// TIA Portal V18 export
ORGANIZATION_BLOCK "10-Main"   // OB1, LAD, ProgramCycle
TITLE = "Main Program / "Main Program Sweep (Cycle)"
{ S7_Optimized_Access := 'TRUE' }
VERSION : 0.1
// stored: AutoNumber true, IsIECCheckEnabled false, SetENOAutomatically false
   VAR_INPUT
      Initial_Call : Bool;   // Initial call of this OB
      Remanence : Bool;   // =True, if remanent data are available
   END_VAR
   VAR_TEMP
      "Temp NormScale" : Real;
      Temp_1 : Bool;
      Temp_2 : Bool;
      "read date val" : DTL;
      "read date out" : Int;
   END_VAR
BEGIN

REGION Network 1: Off, On, Auto Definition
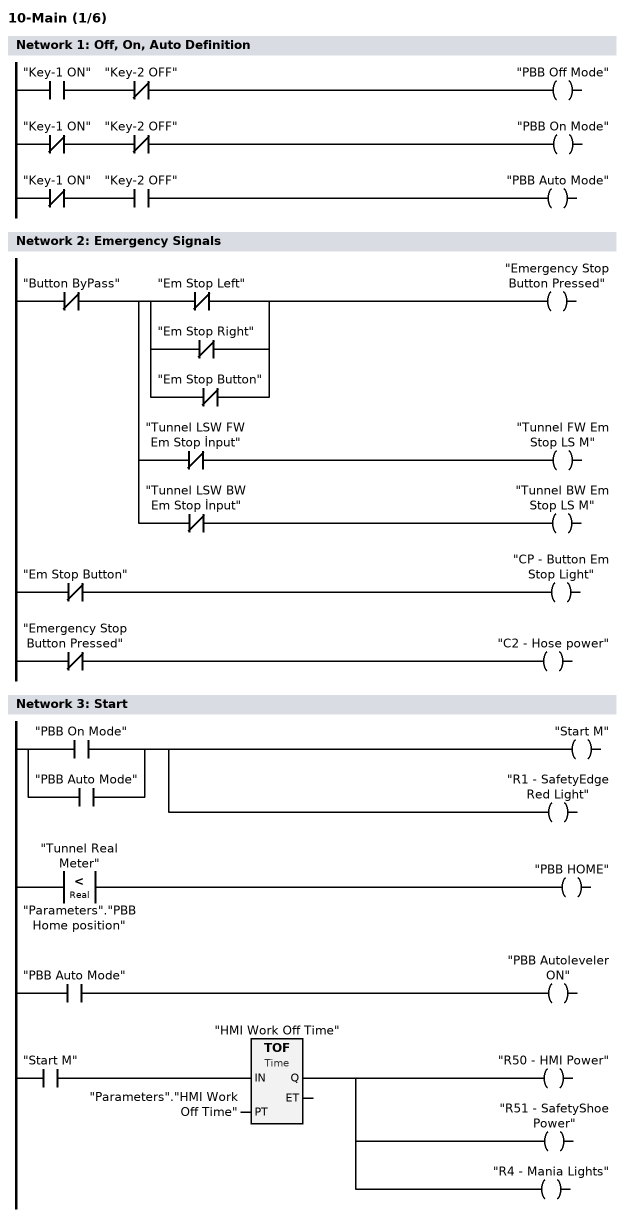
   RUNG wire#powerrail
      Contact( "Key-1 ON" )
      I_Contact( "Key-2 OFF" )
      Coil( "PBB Off Mode" )
   END_RUNG
   RUNG wire#powerrail
      I_Contact( "Key-1 ON" )
      I_Contact( "Key-2 OFF" )
      Coil( "PBB On Mode" )
   END_RUNG
   RUNG wire#powerrail
      I_Contact( "Key-1 ON" )
      Contact( "Key-2 OFF" )
      Coil( "PBB Auto Mode" )
   END_RUNG
   // the same network as SCL:
   "PBB Off Mode" := "Key-1 ON" AND NOT "Key-2 OFF";
   "PBB On Mode" := NOT "Key-1 ON" AND NOT "Key-2 OFF";
   "PBB Auto Mode" := NOT "Key-1 ON" AND "Key-2 OFF";
END_REGION

REGION Network 2: Emergency Signals
   RUNG wire#powerrail
      I_Contact( "Button ByPass" )
      wire#w1
      I_Contact( "Em Stop Left" )
      wire#w2
      Coil( "Emergency Stop Button Pressed" )
   END_RUNG
   RUNG wire#w1
      I_Contact( "Em Stop Right" )
   END_RUNG wire#w2
   RUNG wire#w1
      I_Contact( "Em Stop Button" )
   END_RUNG wire#w2
   RUNG wire#w1
      I_Contact( "Tunnel LSW FW Em Stop İnput" )
      Coil( "Tunnel FW Em Stop LS M" )
   END_RUNG
   RUNG wire#w1
      I_Contact( "Tunnel LSW BW Em Stop İnput" )
      Coil( "Tunnel BW Em Stop LS M" )
   END_RUNG
   RUNG wire#powerrail
      I_Contact( "Em Stop Button" )
      Coil( "CP - Button Em Stop Light" )
   END_RUNG
   RUNG wire#powerrail
      I_Contact( "Emergency Stop Button Pressed" )
      Coil( "C2 - Hose power" )
   END_RUNG
   // the same network as SCL:
   "Emergency Stop Button Pressed" := NOT "Button ByPass" AND (NOT "Em Stop Left" OR NOT "Em Stop Right" OR NOT "Em Stop Button");
   "Tunnel FW Em Stop LS M" := NOT "Button ByPass" AND NOT "Tunnel LSW FW Em Stop İnput";
   "Tunnel BW Em Stop LS M" := NOT "Button ByPass" AND NOT "Tunnel LSW BW Em Stop İnput";
   "CP - Button Em Stop Light" := NOT "Em Stop Button";
   "C2 - Hose power" := NOT "Emergency Stop Button Pressed";
END_REGION

REGION Network 3: Start
   RUNG wire#powerrail
      Contact( "PBB On Mode" )
      wire#w1
      Coil( "Start M" )
   END_RUNG
   RUNG wire#powerrail
      Contact( "PBB Auto Mode" )
   END_RUNG wire#w1
   RUNG wire#w1
      Coil( "R1 - SafetyEdge Red Light" )
   END_RUNG
   RUNG wire#powerrail
      { S7_Templates := "SrcType := Real" } LT_Contact(in1 := "Tunnel Real Meter", in2 := "Parameters"."PBB Home position")
      Coil( "PBB HOME" )
   END_RUNG
   RUNG wire#powerrail
      Contact( "PBB Auto Mode" )
      Coil( "PBB Autoleveler ON" )
   END_RUNG
   RUNG wire#powerrail
      Contact( "Start M" )
      { S7_Templates := "time_type := Time" } "HMI Work Off Time".TOF(pt := "Parameters"."HMI Work Off Time", et =>)
      wire#w2
      Coil( "R50 - HMI Power" )
   END_RUNG
   RUNG wire#w2
      Coil( "R51 - SafetyShoe Power" )
   END_RUNG
   RUNG wire#w2
      Coil( "R4 - Mania Lights" )
   END_RUNG
   // the same network as SCL:
   "Start M" := "PBB On Mode" OR "PBB Auto Mode";
   "R1 - SafetyEdge Red Light" := "Start M";
   "PBB HOME" := "Tunnel Real Meter" < "Parameters"."PBB Home position";
   "PBB Autoleveler ON" := "PBB Auto Mode";
   "HMI Work Off Time".TOF(IN := "Start M", PT := "Parameters"."HMI Work Off Time");
   "R50 - HMI Power" := "HMI Work Off Time".Q;
   "R51 - SafetyShoe Power" := "HMI Work Off Time".Q;
   "R4 - Mania Lights" := "HMI Work Off Time".Q;
END_REGION

REGION Network 4: MC & STO's
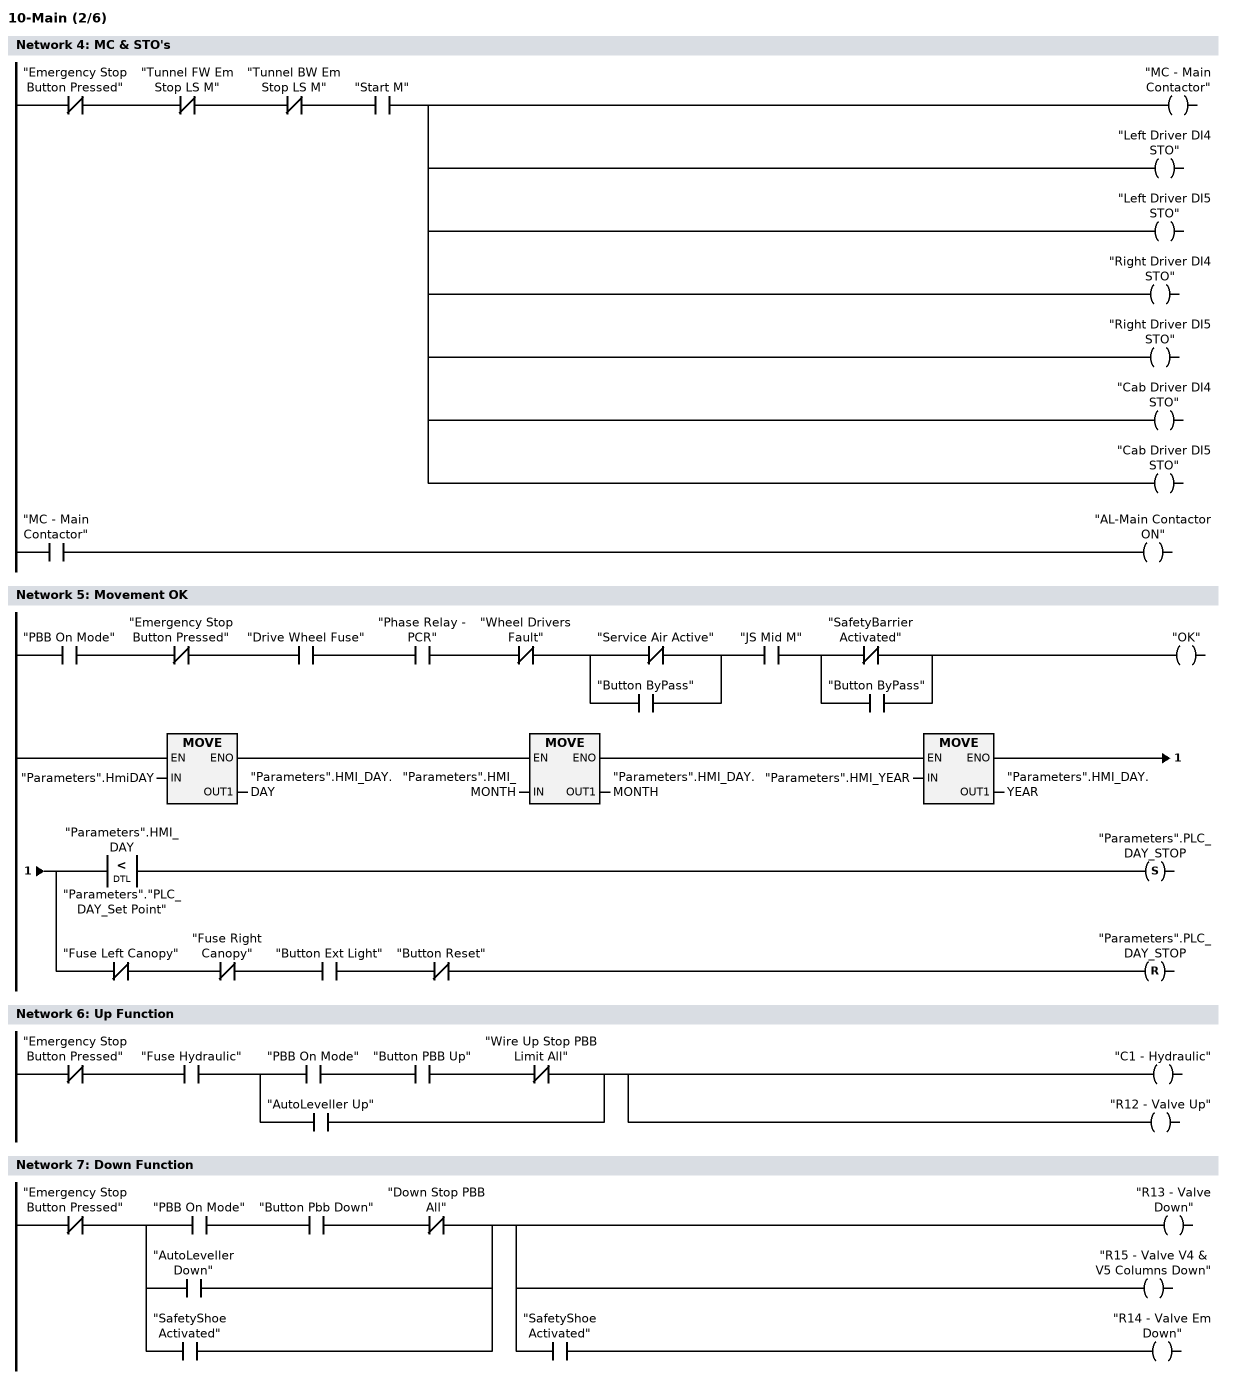
   RUNG wire#powerrail
      I_Contact( "Emergency Stop Button Pressed" )
      I_Contact( "Tunnel FW Em Stop LS M" )
      I_Contact( "Tunnel BW Em Stop LS M" )
      Contact( "Start M" )
      wire#w1
      Coil( "MC - Main Contactor" )
   END_RUNG
   RUNG wire#w1
      Coil( "Left Driver DI4 STO" )
   END_RUNG
   RUNG wire#w1
      Coil( "Left Driver DI5 STO" )
   END_RUNG
   RUNG wire#w1
      Coil( "Right Driver DI4 STO" )
   END_RUNG
   RUNG wire#w1
      Coil( "Right Driver DI5 STO" )
   END_RUNG
   RUNG wire#w1
      Coil( "Cab Driver DI4 STO" )
   END_RUNG
   RUNG wire#w1
      Coil( "Cab Driver DI5 STO" )
   END_RUNG
   RUNG wire#powerrail
      Contact( "MC - Main Contactor" )
      Coil( "AL-Main Contactor ON" )
   END_RUNG
   // the same network as SCL:
   "MC - Main Contactor" := NOT "Emergency Stop Button Pressed" AND NOT "Tunnel FW Em Stop LS M" AND NOT "Tunnel BW Em Stop LS M" AND "Start M";
   "Left Driver DI4 STO" := "MC - Main Contactor";
   "Left Driver DI5 STO" := "MC - Main Contactor";
   "Right Driver DI4 STO" := "MC - Main Contactor";
   "Right Driver DI5 STO" := "MC - Main Contactor";
   "Cab Driver DI4 STO" := "MC - Main Contactor";
   "Cab Driver DI5 STO" := "MC - Main Contactor";
   "AL-Main Contactor ON" := "MC - Main Contactor";
END_REGION

REGION Network 5: Movement OK
   RUNG wire#powerrail
      Contact( "PBB On Mode" )
      I_Contact( "Emergency Stop Button Pressed" )
      Contact( "Drive Wheel Fuse" )
      Contact( "Phase Relay - PCR" )
      I_Contact( "Wheel Drivers Fault" )
      wire#w1
      I_Contact( "Service Air Active" )
      wire#w2
      Contact( "JS Mid M" )
      wire#w3
      I_Contact( "SafetyBarrier Activated" )
      wire#w4
      Coil( "OK" )
   END_RUNG
   RUNG wire#w1
      Contact( "Button ByPass" )
   END_RUNG wire#w2
   RUNG wire#w3
      Contact( "Button ByPass" )
   END_RUNG wire#w4
   RUNG wire#powerrail
      Move(in := "Parameters".HmiDAY, out1 => "Parameters".HMI_DAY.DAY)
      Move(in := "Parameters".HMI_MONTH, out1 => "Parameters".HMI_DAY.MONTH)
      Move(in := "Parameters".HMI_YEAR, out1 => "Parameters".HMI_DAY.YEAR)
      wire#w5
      { S7_Templates := "SrcType := DTL" } LT_Contact(in1 := "Parameters".HMI_DAY, in2 := "Parameters"."PLC_DAY_Set Point")
      S_Coil( "Parameters".PLC_DAY_STOP )
   END_RUNG
   RUNG wire#w5
      I_Contact( "Fuse Left Canopy" )
      I_Contact( "Fuse Right Canopy" )
      Contact( "Button Ext Light" )
      I_Contact( "Button Reset" )
      R_Coil( "Parameters".PLC_DAY_STOP )
   END_RUNG
   // the same network as SCL:
   "OK" := "PBB On Mode" AND NOT "Emergency Stop Button Pressed" AND "Drive Wheel Fuse" AND "Phase Relay - PCR" AND NOT "Wheel Drivers Fault" AND (NOT "Service Air Active" OR "Button ByPass") AND "JS Mid M" AND (NOT "SafetyBarrier Activated" OR "Button ByPass");
   "Parameters".HMI_DAY.DAY := "Parameters".HmiDAY;
   "Parameters".HMI_DAY.MONTH := "Parameters".HMI_MONTH;
   "Parameters".HMI_DAY.YEAR := "Parameters".HMI_YEAR;
   IF "Parameters".HMI_DAY < "Parameters"."PLC_DAY_Set Point" THEN "Parameters".PLC_DAY_STOP := TRUE; END_IF;
   IF NOT "Fuse Left Canopy" AND NOT "Fuse Right Canopy" AND "Button Ext Light" AND NOT "Button Reset" THEN
       "Parameters".PLC_DAY_STOP := FALSE;
   END_IF;
END_REGION

REGION Network 6: Up Function
   RUNG wire#powerrail
      I_Contact( "Emergency Stop Button Pressed" )
      Contact( "Fuse Hydraulic" )
      wire#w1
      Contact( "PBB On Mode" )
      Contact( "Button PBB Up" )
      I_Contact( "Wire Up Stop PBB Limit All" )
      wire#w2
      Coil( "C1 - Hydraulic" )
   END_RUNG
   RUNG wire#w1
      Contact( "AutoLeveller Up" )
   END_RUNG wire#w2
   RUNG wire#w2
      Coil( "R12 - Valve Up" )
   END_RUNG
   // the same network as SCL:
   "C1 - Hydraulic" := NOT "Emergency Stop Button Pressed" AND "Fuse Hydraulic" AND (("PBB On Mode" AND "Button PBB Up" AND NOT "Wire Up Stop PBB Limit All") OR "AutoLeveller Up");
   "R12 - Valve Up" := "C1 - Hydraulic";
END_REGION

REGION Network 7: Down Function
   RUNG wire#powerrail
      I_Contact( "Emergency Stop Button Pressed" )
      wire#w1
      Contact( "PBB On Mode" )
      Contact( "Button Pbb Down" )
      I_Contact( "Down Stop PBB All" )
      wire#w2
      Coil( "R13 - Valve Down" )
   END_RUNG
   RUNG wire#w1
      Contact( "AutoLeveller Down" )
   END_RUNG wire#w2
   RUNG wire#w1
      Contact( "SafetyShoe Activated" )
   END_RUNG wire#w2
   RUNG wire#w2
      Coil( "R15 - Valve V4 & V5 Columns Down" )
   END_RUNG
   RUNG wire#w2
      Contact( "SafetyShoe Activated" )
      Coil( "R14 - Valve Em Down" )
   END_RUNG
   // the same network as SCL:
   "R13 - Valve Down" := NOT "Emergency Stop Button Pressed" AND (("PBB On Mode" AND "Button Pbb Down" AND NOT "Down Stop PBB All") OR "AutoLeveller Down" OR "SafetyShoe Activated");
   "R15 - Valve V4 & V5 Columns Down" := "R13 - Valve Down";
   "R14 - Valve Em Down" := "R13 - Valve Down" AND "SafetyShoe Activated";
END_REGION

REGION Network 8: Faults
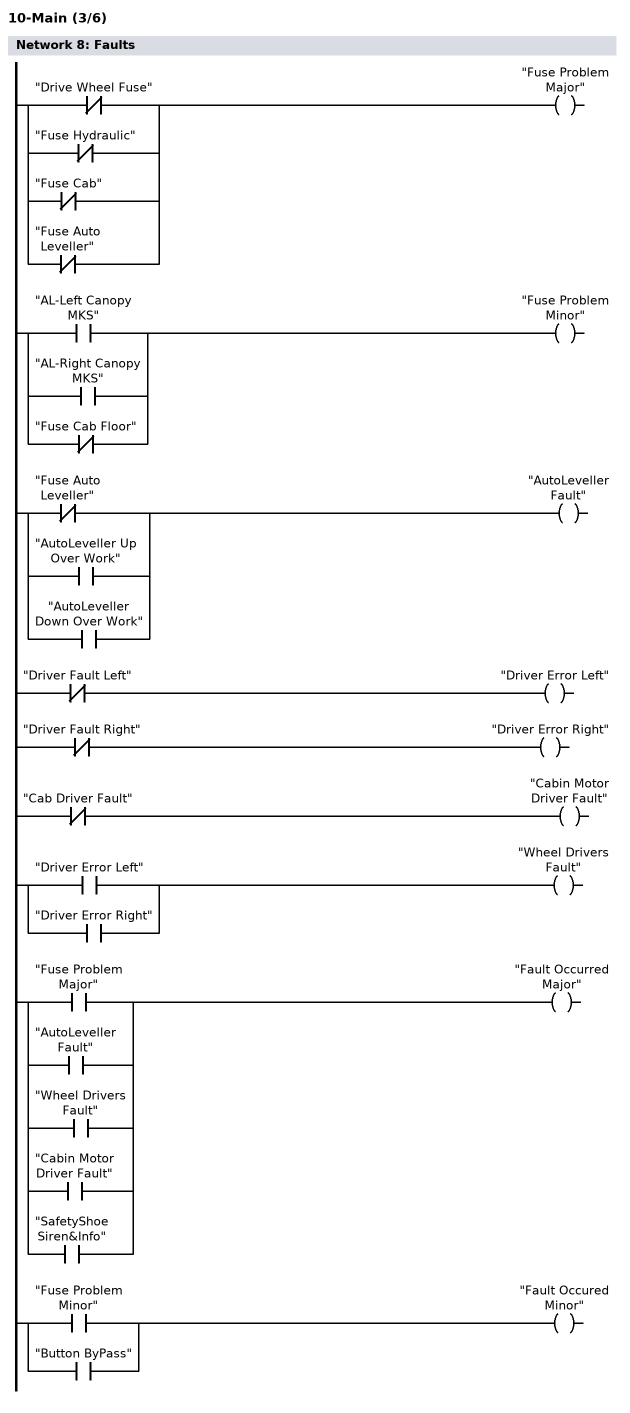
   RUNG wire#powerrail
      I_Contact( "Drive Wheel Fuse" )
      wire#w1
      Coil( "Fuse Problem Major" )
   END_RUNG
   RUNG wire#powerrail
      I_Contact( "Fuse Hydraulic" )
   END_RUNG wire#w1
   RUNG wire#powerrail
      I_Contact( "Fuse Cab" )
   END_RUNG wire#w1
   RUNG wire#powerrail
      I_Contact( "Fuse AutoLeveller" )
   END_RUNG wire#w1
   RUNG wire#powerrail
      Contact( "AL-Left Canopy MKS" )
      wire#w2
      Coil( "Fuse Problem Minor" )
   END_RUNG
   RUNG wire#powerrail
      Contact( "AL-Right Canopy MKS" )
   END_RUNG wire#w2
   RUNG wire#powerrail
      I_Contact( "Fuse Cab Floor" )
   END_RUNG wire#w2
   RUNG wire#powerrail
      I_Contact( "Fuse AutoLeveller" )
      wire#w3
      Coil( "AutoLeveller Fault" )
   END_RUNG
   RUNG wire#powerrail
      Contact( "AutoLeveller Up Over Work" )
   END_RUNG wire#w3
   RUNG wire#powerrail
      Contact( "AutoLeveller Down Over Work" )
   END_RUNG wire#w3
   RUNG wire#powerrail
      I_Contact( "Driver Fault Left" )
      Coil( "Driver Error Left" )
   END_RUNG
   RUNG wire#powerrail
      I_Contact( "Driver Fault Right" )
      Coil( "Driver Error Right" )
   END_RUNG
   RUNG wire#powerrail
      I_Contact( "Cab Driver Fault" )
      Coil( "Cabin Motor Driver Fault" )
   END_RUNG
   RUNG wire#powerrail
      Contact( "Driver Error Left" )
      wire#w4
      Coil( "Wheel Drivers Fault" )
   END_RUNG
   RUNG wire#powerrail
      Contact( "Driver Error Right" )
   END_RUNG wire#w4
   RUNG wire#powerrail
      Contact( "Fuse Problem Major" )
      wire#w5
      Coil( "Fault Occurred Major" )
   END_RUNG
   RUNG wire#powerrail
      Contact( "AutoLeveller Fault" )
   END_RUNG wire#w5
   RUNG wire#powerrail
      Contact( "Wheel Drivers Fault" )
   END_RUNG wire#w5
   RUNG wire#powerrail
      Contact( "Cabin Motor Driver Fault" )
   END_RUNG wire#w5
   RUNG wire#powerrail
      Contact( "SafetyShoe Siren&Info" )
   END_RUNG wire#w5
   RUNG wire#powerrail
      Contact( "Fuse Problem Minor" )
      wire#w6
      Coil( "Fault Occured Minor" )
   END_RUNG
   RUNG wire#powerrail
      Contact( "Button ByPass" )
   END_RUNG wire#w6
   // the same network as SCL:
   "Fuse Problem Major" := NOT "Drive Wheel Fuse" OR NOT "Fuse Hydraulic" OR NOT "Fuse Cab" OR NOT "Fuse AutoLeveller";
   "Fuse Problem Minor" := "AL-Left Canopy MKS" OR "AL-Right Canopy MKS" OR NOT "Fuse Cab Floor";
   "AutoLeveller Fault" := NOT "Fuse AutoLeveller" OR "AutoLeveller Up Over Work" OR "AutoLeveller Down Over Work";
   "Driver Error Left" := NOT "Driver Fault Left";
   "Driver Error Right" := NOT "Driver Fault Right";
   "Cabin Motor Driver Fault" := NOT "Cab Driver Fault";
   "Wheel Drivers Fault" := "Driver Error Left" OR "Driver Error Right";
   "Fault Occurred Major" := "Fuse Problem Major" OR "AutoLeveller Fault" OR "Wheel Drivers Fault" OR "Cabin Motor Driver Fault" OR "SafetyShoe Siren&Info";
   "Fault Occured Minor" := "Fuse Problem Minor" OR "Button ByPass";
END_REGION

REGION Network 9: Reset
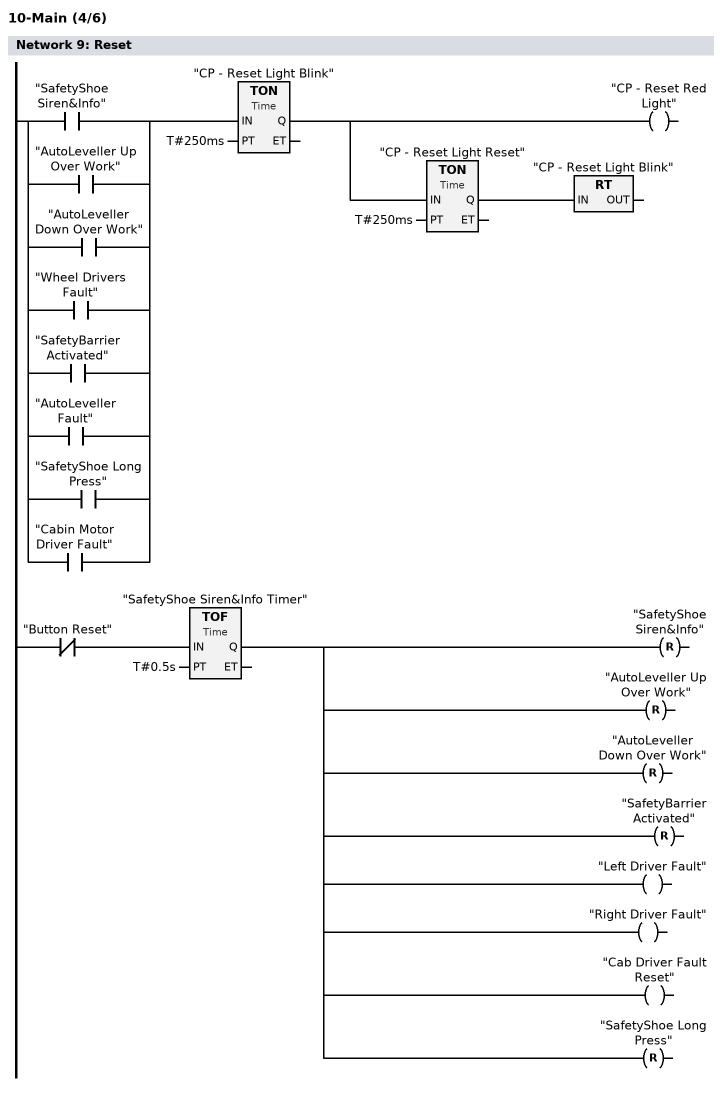
   RUNG wire#powerrail
      Contact( "SafetyShoe Siren&Info" )
      wire#w1
      { S7_Templates := "time_type := Time" } "CP - Reset Light Blink".TON(pt := T#250ms, et =>)
      wire#w2
      Coil( "CP - Reset Red Light" )
   END_RUNG
   RUNG wire#powerrail
      Contact( "AutoLeveller Up Over Work" )
   END_RUNG wire#w1
   RUNG wire#powerrail
      Contact( "AutoLeveller Down Over Work" )
   END_RUNG wire#w1
   RUNG wire#powerrail
      Contact( "Wheel Drivers Fault" )
   END_RUNG wire#w1
   RUNG wire#powerrail
      Contact( "SafetyBarrier Activated" )
   END_RUNG wire#w1
   RUNG wire#powerrail
      Contact( "AutoLeveller Fault" )
   END_RUNG wire#w1
   RUNG wire#powerrail
      Contact( "SafetyShoe Long Press" )
   END_RUNG wire#w1
   RUNG wire#powerrail
      Contact( "Cabin Motor Driver Fault" )
   END_RUNG wire#w1
   RUNG wire#w2
      { S7_Templates := "time_type := Time" } "CP - Reset Light Reset".TON(pt := T#250ms, et =>)
      RT_Coil( "CP - Reset Light Blink" )
   END_RUNG
   RUNG wire#powerrail
      I_Contact( "Button Reset" )
      { S7_Templates := "time_type := Time" } "SafetyShoe Siren&Info Timer".TOF(pt := T#0.5s, et =>)
      wire#w3
      R_Coil( "SafetyShoe Siren&Info" )
   END_RUNG
   RUNG wire#w3
      R_Coil( "AutoLeveller Up Over Work" )
   END_RUNG
   RUNG wire#w3
      R_Coil( "AutoLeveller Down Over Work" )
   END_RUNG
   RUNG wire#w3
      R_Coil( "SafetyBarrier Activated" )
   END_RUNG
   RUNG wire#w3
      Coil( "Left Driver Fault" )
   END_RUNG
   RUNG wire#w3
      Coil( "Right Driver Fault" )
   END_RUNG
   RUNG wire#w3
      Coil( "Cab Driver Fault Reset" )
   END_RUNG
   RUNG wire#w3
      R_Coil( "SafetyShoe Long Press" )
   END_RUNG
   // the same network as SCL:
   "CP - Reset Light Blink".TON(IN := "SafetyShoe Siren&Info" OR "AutoLeveller Up Over Work" OR "AutoLeveller Down Over Work" OR "Wheel Drivers Fault" OR "SafetyBarrier Activated" OR "AutoLeveller Fault" OR "SafetyShoe Long Press" OR "Cabin Motor Driver Fault",
                           PT := T#250ms);
   "CP - Reset Red Light" := "CP - Reset Light Blink".Q;
   "CP - Reset Light Reset".TON(IN := "CP - Reset Light Blink".Q, PT := T#250ms);
   IF "CP - Reset Light Reset".Q THEN RESET_TIMER("CP - Reset Light Blink"); END_IF;
   "SafetyShoe Siren&Info Timer".TOF(IN := NOT "Button Reset", PT := T#0.5s);
   IF "SafetyShoe Siren&Info Timer".Q THEN
       "SafetyShoe Siren&Info" := FALSE;
       "AutoLeveller Up Over Work" := FALSE;
       "AutoLeveller Down Over Work" := FALSE;
       "SafetyBarrier Activated" := FALSE;
   END_IF;
   "Left Driver Fault" := "SafetyShoe Siren&Info Timer".Q;
   "Right Driver Fault" := "SafetyShoe Siren&Info Timer".Q;
   "Cab Driver Fault Reset" := "SafetyShoe Siren&Info Timer".Q;
   IF "SafetyShoe Siren&Info Timer".Q THEN "SafetyShoe Long Press" := FALSE; END_IF;
END_REGION

REGION Network 10: Indicators & Warning Lights
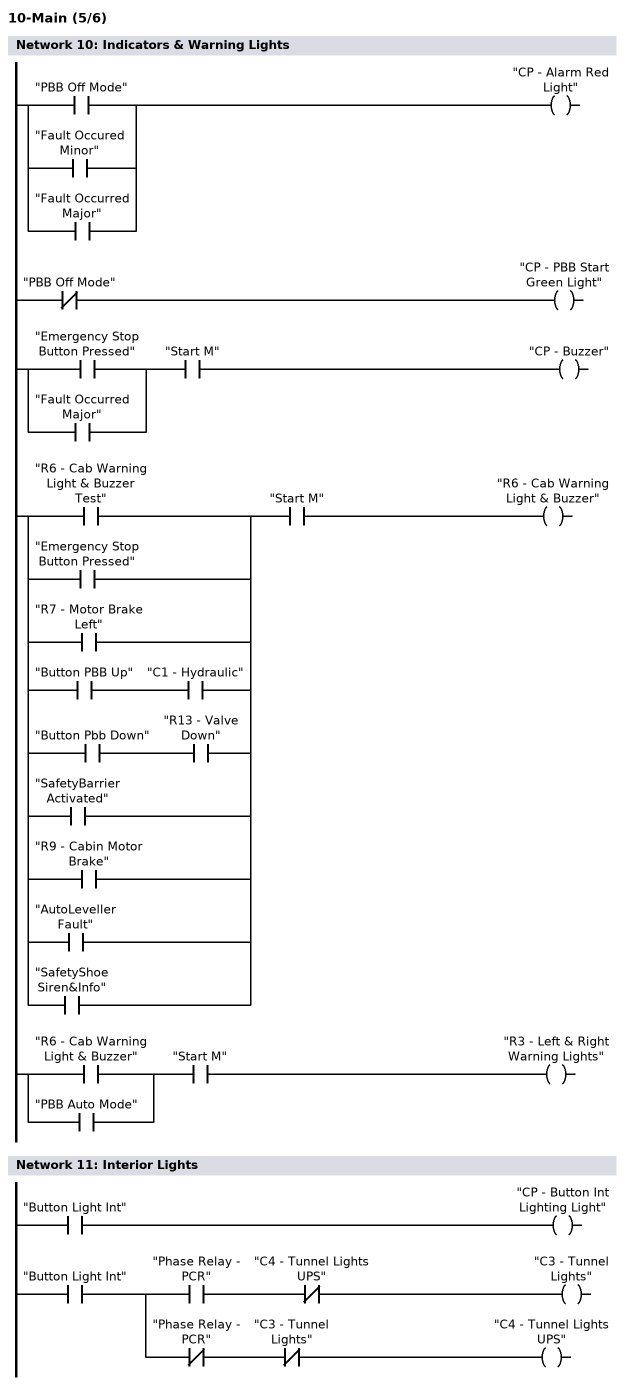
   RUNG wire#powerrail
      Contact( "PBB Off Mode" )
      wire#w1
      Coil( "CP - Alarm Red Light" )
   END_RUNG
   RUNG wire#powerrail
      Contact( "Fault Occured Minor" )
   END_RUNG wire#w1
   RUNG wire#powerrail
      Contact( "Fault Occurred Major" )
   END_RUNG wire#w1
   RUNG wire#powerrail
      I_Contact( "PBB Off Mode" )
      Coil( "CP - PBB Start Green Light" )
   END_RUNG
   RUNG wire#powerrail
      Contact( "Emergency Stop Button Pressed" )
      wire#w2
      Contact( "Start M" )
      Coil( "CP - Buzzer" )
   END_RUNG
   RUNG wire#powerrail
      Contact( "Fault Occurred Major" )
   END_RUNG wire#w2
   RUNG wire#powerrail
      Contact( "R6 - Cab Warning Light & Buzzer Test" )
      wire#w3
      Contact( "Start M" )
      Coil( "R6 - Cab Warning Light & Buzzer" )
   END_RUNG
   RUNG wire#powerrail
      Contact( "Emergency Stop Button Pressed" )
   END_RUNG wire#w3
   RUNG wire#powerrail
      Contact( "R7 - Motor Brake Left" )
   END_RUNG wire#w3
   RUNG wire#powerrail
      Contact( "Button PBB Up" )
      Contact( "C1 - Hydraulic" )
   END_RUNG wire#w3
   RUNG wire#powerrail
      Contact( "Button Pbb Down" )
      Contact( "R13 - Valve Down" )
   END_RUNG wire#w3
   RUNG wire#powerrail
      Contact( "SafetyBarrier Activated" )
   END_RUNG wire#w3
   RUNG wire#powerrail
      Contact( "R9 - Cabin Motor Brake" )
   END_RUNG wire#w3
   RUNG wire#powerrail
      Contact( "AutoLeveller Fault" )
   END_RUNG wire#w3
   RUNG wire#powerrail
      Contact( "SafetyShoe Siren&Info" )
   END_RUNG wire#w3
   RUNG wire#powerrail
      Contact( "R6 - Cab Warning Light & Buzzer" )
      wire#w4
      Contact( "Start M" )
      Coil( "R3 - Left & Right Warning Lights" )
   END_RUNG
   RUNG wire#powerrail
      Contact( "PBB Auto Mode" )
   END_RUNG wire#w4
   // the same network as SCL:
   "CP - Alarm Red Light" := "PBB Off Mode" OR "Fault Occured Minor" OR "Fault Occurred Major";
   "CP - PBB Start Green Light" := NOT "PBB Off Mode";
   "CP - Buzzer" := ("Emergency Stop Button Pressed" OR "Fault Occurred Major") AND "Start M";
   "R6 - Cab Warning Light & Buzzer" := ("R6 - Cab Warning Light & Buzzer Test" OR "Emergency Stop Button Pressed" OR "R7 - Motor Brake Left" OR ("Button PBB Up" AND "C1 - Hydraulic") OR ("Button Pbb Down" AND "R13 - Valve Down") OR "SafetyBarrier Activated" OR "R9 - Cabin Motor Brake" OR "AutoLeveller Fault" OR "SafetyShoe Siren&Info") AND "Start M";
   "R3 - Left & Right Warning Lights" := ("R6 - Cab Warning Light & Buzzer" OR "PBB Auto Mode") AND "Start M";
END_REGION

REGION Network 11: Interior Lights
   RUNG wire#powerrail
      Contact( "Button Light Int" )
      Coil( "CP - Button Int Lighting Light" )
   END_RUNG
   RUNG wire#powerrail
      Contact( "Button Light Int" )
      wire#w1
      Contact( "Phase Relay - PCR" )
      I_Contact( "C4 - Tunnel Lights UPS" )
      Coil( "C3 - Tunnel Lights" )
   END_RUNG
   RUNG wire#w1
      I_Contact( "Phase Relay - PCR" )
      I_Contact( "C3 - Tunnel Lights" )
      Coil( "C4 - Tunnel Lights UPS" )
   END_RUNG
   // the same network as SCL:
   "CP - Button Int Lighting Light" := "Button Light Int";
   "C3 - Tunnel Lights" := "Button Light Int" AND "Phase Relay - PCR" AND NOT "C4 - Tunnel Lights UPS";
   "C4 - Tunnel Lights UPS" := "Button Light Int" AND NOT "Phase Relay - PCR" AND NOT "C3 - Tunnel Lights";
END_REGION

REGION Network 12: Exterior Lights
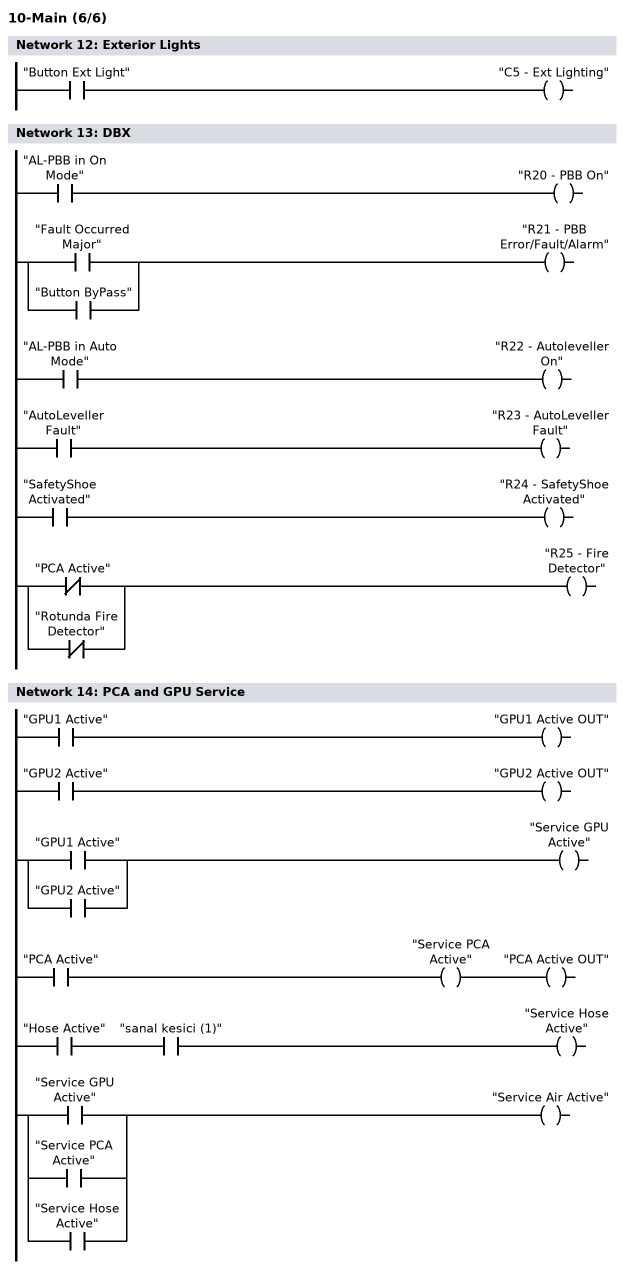
   RUNG wire#powerrail
      Contact( "Button Ext Light" )
      Coil( "C5 - Ext Lighting" )
   END_RUNG
   // the same network as SCL:
   "C5 - Ext Lighting" := "Button Ext Light";
END_REGION

REGION Network 13: DBX
   RUNG wire#powerrail
      Contact( "AL-PBB in On Mode" )
      Coil( "R20 - PBB On" )
   END_RUNG
   RUNG wire#powerrail
      Contact( "Fault Occurred Major" )
      wire#w1
      Coil( "R21 - PBB Error/Fault/Alarm" )
   END_RUNG
   RUNG wire#powerrail
      Contact( "Button ByPass" )
   END_RUNG wire#w1
   RUNG wire#powerrail
      Contact( "AL-PBB in Auto Mode" )
      Coil( "R22 - Autoleveller On" )
   END_RUNG
   RUNG wire#powerrail
      Contact( "AutoLeveller Fault" )
      Coil( "R23 - AutoLeveller Fault" )
   END_RUNG
   RUNG wire#powerrail
      Contact( "SafetyShoe Activated" )
      Coil( "R24 - SafetyShoe Activated" )
   END_RUNG
   RUNG wire#powerrail
      I_Contact( "PCA Active" )
      wire#w2
      Coil( "R25 - Fire Detector" )
   END_RUNG
   RUNG wire#powerrail
      I_Contact( "Rotunda Fire Detector" )
   END_RUNG wire#w2
   // the same network as SCL:
   "R20 - PBB On" := "AL-PBB in On Mode";
   "R21 - PBB Error/Fault/Alarm" := "Fault Occurred Major" OR "Button ByPass";
   "R22 - Autoleveller On" := "AL-PBB in Auto Mode";
   "R23 - AutoLeveller Fault" := "AutoLeveller Fault";
   "R24 - SafetyShoe Activated" := "SafetyShoe Activated";
   "R25 - Fire Detector" := NOT "PCA Active" OR NOT "Rotunda Fire Detector";
END_REGION

REGION Network 14: PCA and GPU Service
   RUNG wire#powerrail
      Contact( "GPU1 Active" )
      Coil( "GPU1 Active OUT" )
   END_RUNG
   RUNG wire#powerrail
      Contact( "GPU2 Active" )
      Coil( "GPU2 Active OUT" )
   END_RUNG
   RUNG wire#powerrail
      Contact( "GPU1 Active" )
      wire#w1
      Coil( "Service GPU Active" )
   END_RUNG
   RUNG wire#powerrail
      Contact( "GPU2 Active" )
   END_RUNG wire#w1
   RUNG wire#powerrail
      Contact( "PCA Active" )
      Coil( "Service PCA Active" )
      Coil( "PCA Active OUT" )
   END_RUNG
   RUNG wire#powerrail
      Contact( "Hose Active" )
      Contact( "sanal kesici (1)" )
      Coil( "Service Hose Active" )
   END_RUNG
   RUNG wire#powerrail
      Contact( "Service GPU Active" )
      wire#w2
      Coil( "Service Air Active" )
   END_RUNG
   RUNG wire#powerrail
      Contact( "Service PCA Active" )
   END_RUNG wire#w2
   RUNG wire#powerrail
      Contact( "Service Hose Active" )
   END_RUNG wire#w2
   // the same network as SCL:
   "GPU1 Active OUT" := "GPU1 Active";
   "GPU2 Active OUT" := "GPU2 Active";
   "Service GPU Active" := "GPU1 Active" OR "GPU2 Active";
   "Service PCA Active" := "PCA Active";
   "PCA Active OUT" := "PCA Active";
   "Service Hose Active" := "Hose Active" AND "sanal kesici (1)";
   "Service Air Active" := "Service GPU Active" OR "Service PCA Active" OR "Service Hose Active";
END_REGION
END_ORGANIZATION_BLOCK
